Staubli VAL3: uListTRSF.pgx

program uListTRSF(trsf& x_TRSF[] (dimensions=1), string& x_sTRSF[] (dimensions=1))
  local num l_i
begin
  call up:listSetSize(0,7,38,4)
  call up:listCreate("")
  for l_i=0 to 3
    call ut:_trsf2String(x_TRSF[l_i],"Location p"+toString("",l_i),"",7,x_sTRSF[l_i])
  endFor
  call up:listAdd(x_sTRSF)
  call up:listUpdate(0)
end
